INTERFACE ITF_Component1 EXTENDS ITF_BaseComponent

END_INTERFACE

(* stored: Version 1.1.0.1
   Itf ITF_Component1: Id {715b39ee-2c73-0f2b-0f2b-d76dd1c76701} *)
